(* Logix 5000 project; controller inz_PD_LK vendor 1 type 14 code 285 rev 34.11; software revision 34.01 *)

TASK MainTask (continuous, watchdog 500 ms) : Paleczka_silnik, Dzwonki_silnik, Paleczka_note_move, Dzwonki_belt_move, buttons, status, TIMER, Lights, oda, kolejnosc, dzwieki

MODULES
   Local : vendor 1 type 14 code 285 (5069 0, rev 34.11)
      serwowzmacniacz : vendor 1 type 45 code 1 (Ethernet 192.168.1.26, rev 5.2, AMotionDiagnostics RPI 1 ms)
      serwowzmacniacz2 : vendor 1 type 45 code 1 (Ethernet 192.168.1.27, rev 5.2, AMotionDiagnostics RPI 1 ms)
      Input : 5069-IB16 (5069 1, rev 2.1, StandardDataDriven RPI 5 ms)
      Output : 5069-OB16 (5069 2, rev 3.1, StandardDataDriven RPI 5 ms)
      Wyspa : 1734-AENTR (Ethernet 192.168.1.24, rev 5.12, Output RPI 20 ms)
         IB8 : 1734-IB8 (PointIO 3, rev 3.1)
         IB8_2 : 1734-IB8 (PointIO 4, rev 3.1)
         IE8C : vendor 1 type 115 code 210 (PointIO 6, rev 3.1, Input RPI 80 ms)
         OB8 : 1734-OB8 (PointIO 1, rev 3.1)
         OB8_2 : 1734-OB8 (PointIO 2, rev 3.1)
         OE4C : vendor 1 type 115 code 211 (PointIO 5, rev 3.1, Output RPI 80 ms)
END_MODULES

VAR_GLOBAL   (* controller tags *)
   all_rise : BOOL;
   auto_belt : BOOL;
   auto_mode : ALIAS FOR Local:1:I.Pt09.Data;
   auto_note : BOOL;
   belt_degree : DINT := 58;
   belt_finish : BOOL;
   D_JOG_Axis_OFF : BOOL := 1;
   D_JOG_Axis_ON : BOOL;
   D_motor_start : BOOL;
   D_motor_stop : BOOL := 1;
   degree : DINT := 20;
   dzwiek : DINT[50] := ([1] := 29, [2] := 29, [4] := -29, [5] := -29, [6] := -29, [7] := -29, [9] := 29, [10] := 29, [12] := -29, [14] := 29, [16] := 29, [17] := 29, [19] := -29, [20] := -29, [21] := -29, [22] := -29, [24] := 29, [25] := 29, [26] := -29, [27] := -29);
   Dzwonki : AXIS_CIP_DRIVE;
   Estop_button : ALIAS FOR Local:1:I.Pt00.Data;
   forced_OFF : BOOL;
   forced_ON : BOOL := 1;
   go_down : BOOL;
   go_left : ALIAS FOR Wyspa:3:I.5;
   go_right : ALIAS FOR Local:1:I.Pt02.Data;
   go_up : BOOL;
   green_lamp : ALIAS FOR Local:2:O.Pt13.Data;
   L_R_switch : ALIAS FOR Local:1:I.Pt10.Data;
   Motion : MOTION_GROUP;
   MotionControlMAFR_D : MOTION_INSTRUCTION := (FLAGS := 570425344, DN := 1, STATE := 1);
   MotionControlMAFR_P : MOTION_INSTRUCTION := (FLAGS := 570425344, DN := 1, STATE := 1);
   MotionControlMAH : MOTION_INSTRUCTION := (FLAGS := 33554432);
   MotionControlMAJ_P : MOTION_INSTRUCTION := (FLAGS := 301989888, ER := 1, ERR := 5);
   MotionControlMAM : MOTION_INSTRUCTION := (FLAGS := 570425344, DN := 1);
   MotionControlMAM2 : MOTION_INSTRUCTION := (FLAGS := 704643072, DN := 1, PC := 1);
   MotionControlMAM3 : MOTION_INSTRUCTION := (FLAGS := 704643072, DN := 1, PC := 1);
   MotionControlMAM4 : MOTION_INSTRUCTION := (FLAGS := 33554432);
   MotionControlMAM5 : MOTION_INSTRUCTION := (FLAGS := 704643072, DN := 1, PC := 1);
   MotionControlMAS_D : MOTION_INSTRUCTION := (FLAGS := -1442840576, EN := 1, DN := 1, PC := 1);
   MotionControlMAS_P : MOTION_INSTRUCTION := (FLAGS := -1442840576, EN := 1, DN := 1, PC := 1);
   MotionControlOFF_D : MOTION_INSTRUCTION := (FLAGS := -1577058304, EN := 1, DN := 1, STATUS := 2, STATE := 1);
   MotionControlOFF_P : MOTION_INSTRUCTION := (FLAGS := -1577058304, EN := 1, DN := 1, STATUS := 2, STATE := 1);
   MotionControlON_D : MOTION_INSTRUCTION := (FLAGS := 570425344, DN := 1, STATE := 1);
   MotionControlON_P : MOTION_INSTRUCTION := (FLAGS := 570425344, DN := 1, STATE := 1);
   move_belt : BOOL;
   neg_belt_degree : DINT := -58;
   neg_degree : INT := -20;
   OSR_auto_belt : BOOL;
   OSR_auto_note : BOOL;
   OSR_belt_ready : BOOL;
   OSR_D_motor_start : BOOL;
   OSR_D_motor_stop : BOOL;
   OSR_forced_OFF : BOOL;
   OSR_forced_ON : BOOL;
   OSR_moved : BOOL;
   OSR_P_motor_start : BOOL;
   OSR_P_motor_stop : BOOL;
   OSR_start_now : BOOL;
   OSR_starting_ON : BOOL;
   P_JOG_Axis_OFF : BOOL := 1;
   P_JOG_Axis_ON : BOOL;
   P_motor_start : BOOL;
   P_motor_stop : BOOL := 1;
   Paleczka : AXIS_CIP_DRIVE;
   play_note : BOOL;
   play_note_rise : BOOL;
   PULSE_1Hz : BOOL := 1;
   PULSE_2Hz : BOOL := 1;
   ready : BOOL;
   red_lamp : ALIAS FOR Local:2:O.Pt15.Data;
   reset : BOOL;
   reset_button : ALIAS FOR Local:1:I.Pt07.Data;
   stand_by : BOOL;
   start : BOOL; {access None}
   start_button : ALIAS FOR Local:1:I.Pt05.Data;
   start_degree : DINT := 20;
   start_now : BOOL;
   starting_ON : BOOL := 1;
   stop : BOOL := 1; {access None}
   switch_OFF : ALIAS FOR Local:1:I.Pt08.Data;
   switch_ON : ALIAS FOR Local:1:I.Pt09.Data;
   TIMER1N : TIMER := (PRE := 100);
   TIMER2N : TIMER := (PRE := 200);
   uderzenie : DINT[50] := ([0] := 20, [1] := 20, [2] := 20, [3] := 20, [4] := 20, [5] := 20);
   yellow_lamp : ALIAS FOR Local:2:O.Pt14.Data;
END_VAR

PROGRAM buttons   (* main routine buttons *)

ROUTINE buttons   (* ladder *)
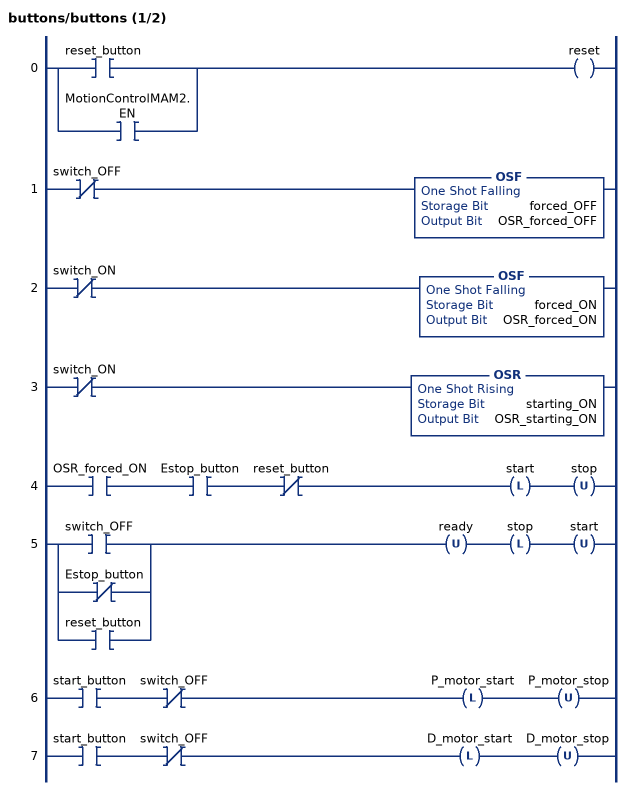
   0: [XIC(reset_button) ,XIC(MotionControlMAM2.EN) ]OTE(reset);
   1: XIO(switch_OFF)OSF(forced_OFF,OSR_forced_OFF);
   2: XIO(switch_ON)OSF(forced_ON,OSR_forced_ON);
   3: XIO(switch_ON)OSR(starting_ON,OSR_starting_ON);
   4: XIC(OSR_forced_ON)XIC(Estop_button)XIO(reset_button)OTL(start)OTU(stop);
   5: [XIC(switch_OFF) ,[XIO(Estop_button) ,XIC(reset_button) ] ]OTU(ready)OTL(stop)OTU(start);
   6: XIC(start_button)XIO(switch_OFF)OTL(P_motor_start)OTU(P_motor_stop);
   7: XIC(start_button)XIO(switch_OFF)OTL(D_motor_start)OTU(D_motor_stop);
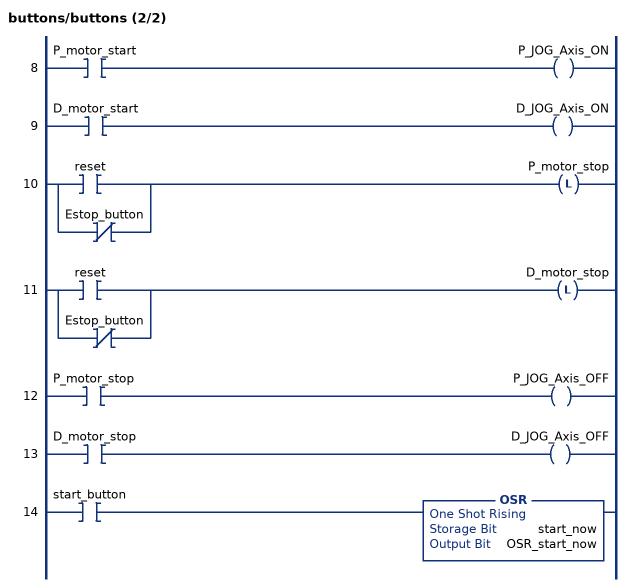
   8: XIC(P_motor_start)OTE(P_JOG_Axis_ON);
   9: XIC(D_motor_start)OTE(D_JOG_Axis_ON);
   10: [XIC(reset) ,XIO(Estop_button) ]OTL(P_motor_stop);
   11: [XIC(reset) ,XIO(Estop_button) ]OTL(D_motor_stop);
   12: XIC(P_motor_stop)OTE(P_JOG_Axis_OFF);
   13: XIC(D_motor_stop)OTE(D_JOG_Axis_OFF);
   14: XIC(start_button)OSR(start_now,OSR_start_now);
END_ROUTINE
END_PROGRAM

PROGRAM dzwieki   (* main routine dzwieki *)

ROUTINE dzwieki   (* structured text *)
   // "Oda do radości" zaczynając od E
   dzwiek[0] := 0;    //E <- druga nuta
   dzwiek[1] := 29;   //F
   dzwiek[2] := 29;   //G
   dzwiek[3] := 0;    //G
   dzwiek[4] := -29;  //F
   dzwiek[5] := -29;  //E
   dzwiek[6] := -29;  //D
   dzwiek[7] := -29;  //C
   dzwiek[8] := 0;    //C
   dzwiek[9] := 29;   //D
   dzwiek[10] := 29;  //E
   dzwiek[11] := 0;   //E
   dzwiek[12] := -29; //D
   dzwiek[13] := 0;   //D
   dzwiek[14] := 29;  //E
   dzwiek[15] := 0;   //E
   dzwiek[16] := 29;  //F
   dzwiek[17] := 29;  //G
   dzwiek[18] := 0;   //G
   dzwiek[19] := -29; //F
   dzwiek[20] := -29; //E
   dzwiek[21] := -29; //D
   dzwiek[22] := -29; //C
   dzwiek[23] := 0;   //C
   dzwiek[24] := 29;  //D
   dzwiek[25] := 29;  //E
   dzwiek[26] := -29; //D
   dzwiek[27] := -29; //C
   dzwiek[28] := 0;   //C
END_ROUTINE
END_PROGRAM

PROGRAM Dzwonki_belt_move   (* main routine belt_move *)
VAR
   acc : DINT := 2000;
   belt_moving : DINT := 30;
   belt_ready : BOOL;
   CTU1 : COUNTER := (ACC := 30, DN := 1);
   jerk : DINT := 14;
   odl : DINT := 58;
   speed : DINT := 10000;
END_VAR

ROUTINE belt_move   (* ladder *)
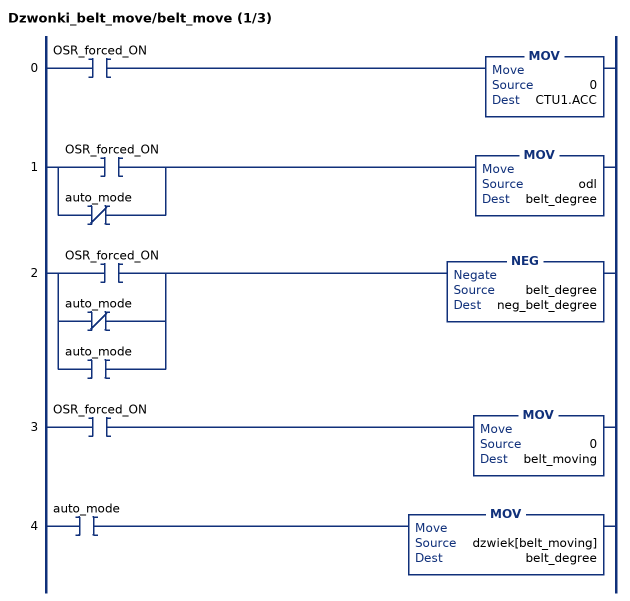
   0: XIC(OSR_forced_ON)MOV(0,CTU1.ACC);
   1: [XIC(OSR_forced_ON) ,XIO(auto_mode) ]MOV(odl,belt_degree);
   2: [XIC(OSR_forced_ON) ,[XIO(auto_mode) ,XIC(auto_mode) ] ]NEG(belt_degree,neg_belt_degree);
   3: XIC(OSR_forced_ON)MOV(0,belt_moving);
   4: XIC(auto_mode)MOV(dzwiek[belt_moving],belt_degree);
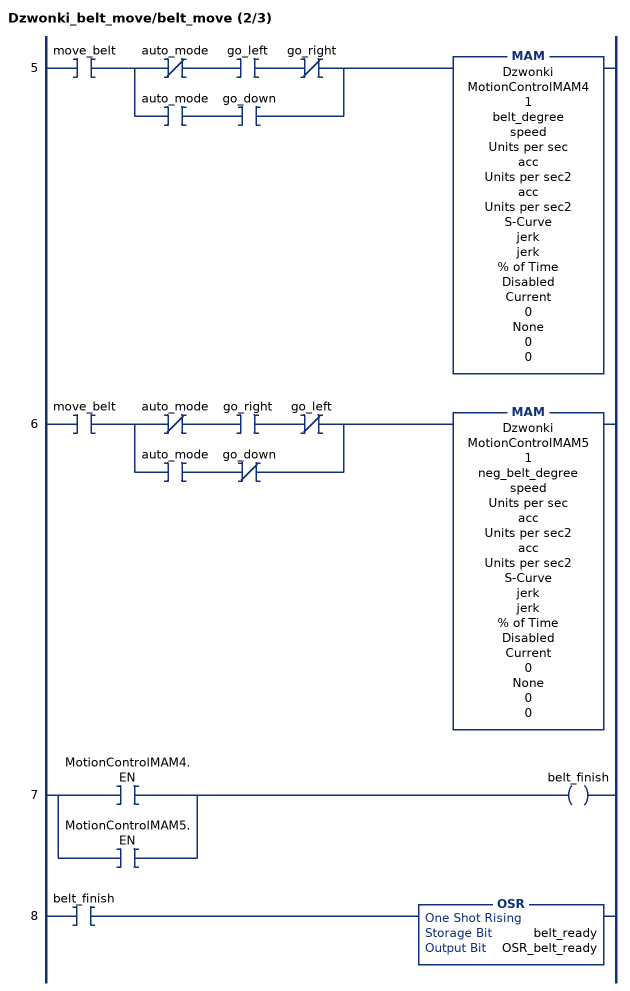
   5: XIC(move_belt)[XIO(auto_mode) XIC(go_left) XIO(go_right) ,XIC(auto_mode) XIC(go_down) ]MAM(Dzwonki,MotionControlMAM4,1,belt_degree,speed,Units per sec,acc,Units per sec2,acc,Units per sec2,S-Curve,jerk,jerk,% of Time,Disabled,Current,0,None,0,0);
   6: XIC(move_belt)[XIO(auto_mode) XIC(go_right) XIO(go_left) ,XIC(auto_mode) XIO(go_down) ]MAM(Dzwonki,MotionControlMAM5,1,neg_belt_degree,speed,Units per sec,acc,Units per sec2,acc,Units per sec2,S-Curve,jerk,jerk,% of Time,Disabled,Current,0,None,0,0);
   7: [XIC(MotionControlMAM4.EN) ,XIC(MotionControlMAM5.EN) ]OTE(belt_finish);
   8: XIC(belt_finish)OSR(belt_ready,OSR_belt_ready);
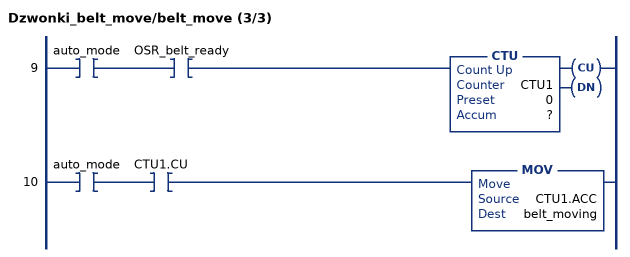
   9: XIC(auto_mode)XIC(OSR_belt_ready)CTU(CTU1,?,?);
   10: XIC(auto_mode)XIC(CTU1.CU)MOV(CTU1.ACC,belt_moving);
END_ROUTINE
END_PROGRAM

PROGRAM Dzwonki_silnik   (* main routine MainRoutine *)

ROUTINE MainRoutine   (* ladder *)
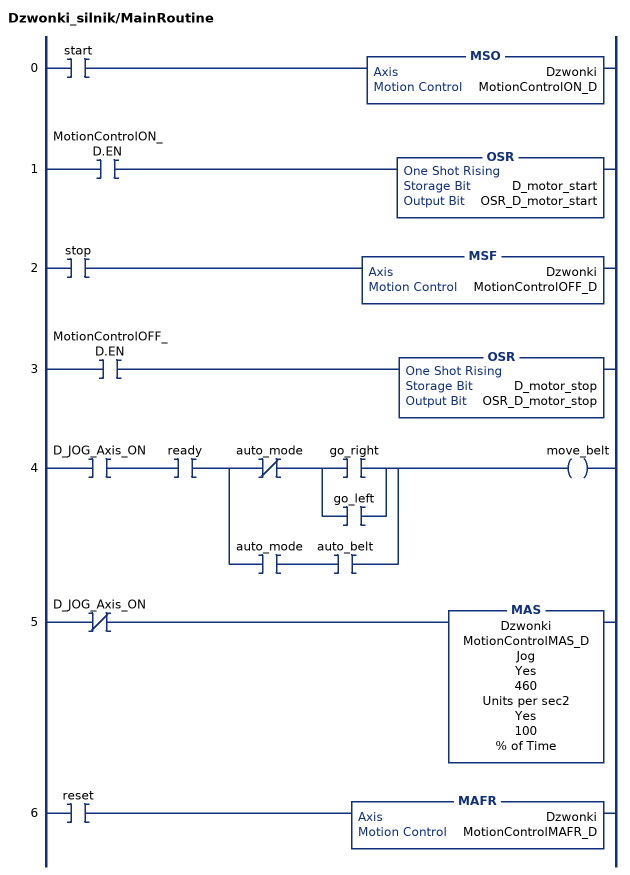
   0: XIC(start)MSO(Dzwonki,MotionControlON_D);
   1: XIC(MotionControlON_D.EN)OSR(D_motor_start,OSR_D_motor_start);
   2: XIC(stop)MSF(Dzwonki,MotionControlOFF_D);
   3: XIC(MotionControlOFF_D.EN)OSR(D_motor_stop,OSR_D_motor_stop);
   4: XIC(D_JOG_Axis_ON)XIC(ready)[XIO(auto_mode) [XIC(go_right) ,XIC(go_left) ] ,XIC(auto_mode) XIC(auto_belt) ]OTE(move_belt);
   5: XIO(D_JOG_Axis_ON)MAS(Dzwonki,MotionControlMAS_D,Jog,Yes,460,Units per sec2,Yes,100,% of Time);
   6: XIC(reset)MAFR(Dzwonki,MotionControlMAFR_D);
END_ROUTINE
END_PROGRAM

PROGRAM kolejnosc   (* main routine kolejnosc *)

ROUTINE kolejnosc   (* structured text *)
   uderzenie[0] := 20;
   uderzenie[1] := 20;
   uderzenie[2] := 20;
   uderzenie[3] := 20;
   uderzenie[4] := 20;
   uderzenie[5] := 20;
   
END_ROUTINE
END_PROGRAM

PROGRAM Lights   (* main routine Lights *)
VAR
   OSR_yellow_ON : BOOL;
   yellow_ON : BOOL;
END_VAR

ROUTINE Lights   (* ladder *)
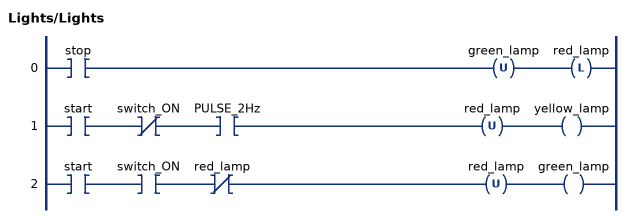
   0: XIC(stop)OTU(green_lamp)OTL(red_lamp);
   1: XIC(start)XIO(switch_ON)XIC(PULSE_2Hz)OTU(red_lamp)OTE(yellow_lamp);
   2: XIC(start)XIC(switch_ON)XIO(red_lamp)OTU(red_lamp)OTE(green_lamp);
END_ROUTINE
END_PROGRAM

PROGRAM oda   (* main routine oda *)
VAR
   CTU1 : COUNTER := (PRE := 1, ACC := 30, CD := 1, DN := 1);
   CTU1_CU : BOOL;
   CTU2 : COUNTER := (PRE := 5);
   even_odd : DINT;
   is_finished : BOOL;
   LCONS_INIT : INT;
   ONS_auto_belt : BOOL;
   ONS_auto_note : BOOL;
   ONS_is_finished : BOOL;
   OSR_CTU1_CU : BOOL;
   OSR_timer1_ready : BOOL;
   OSR_timer2_ready : BOOL;
   repeats : DINT;
   STEP : INT;
   timer1_ready : BOOL;
   TIMER1O : TIMER := (PRE := 100);
   timer2_ready : BOOL;
   TIMER2O : TIMER := (PRE := 100);
   TON1 : TIMER := (PRE := 50);
END_VAR

ROUTINE oda   (* ladder *)
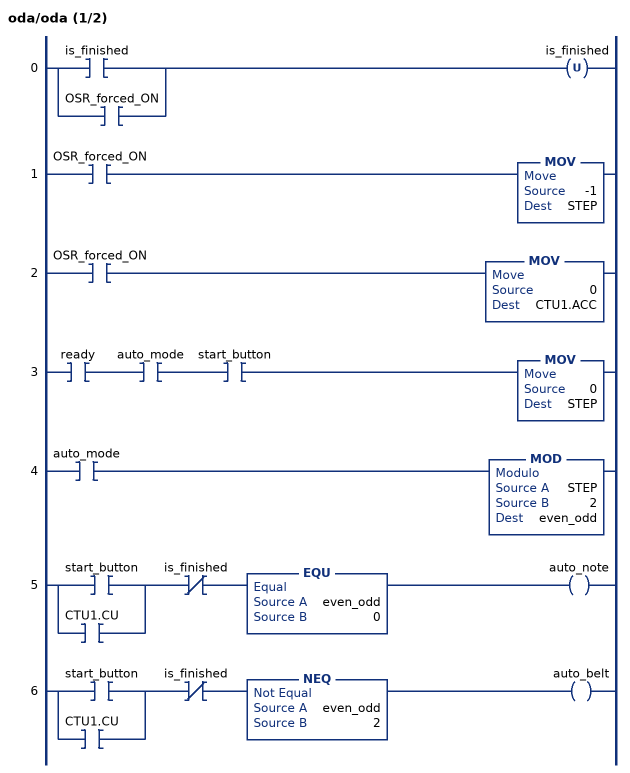
   0: [XIC(is_finished) ,XIC(OSR_forced_ON) ]OTU(is_finished);
   1: XIC(OSR_forced_ON)MOV(-1,STEP);
   2: XIC(OSR_forced_ON)MOV(0,CTU1.ACC);
   3: XIC(ready)XIC(auto_mode)XIC(start_button)MOV(0,STEP);
   4: XIC(auto_mode)MOD(STEP,2,even_odd);
   5: [XIC(start_button) ,XIC(CTU1.CU) ]XIO(is_finished)EQU(even_odd,0)OTE(auto_note);
   6: [XIC(start_button) ,XIC(CTU1.CU) ]XIO(is_finished)NEQ(even_odd,2)OTE(auto_belt);
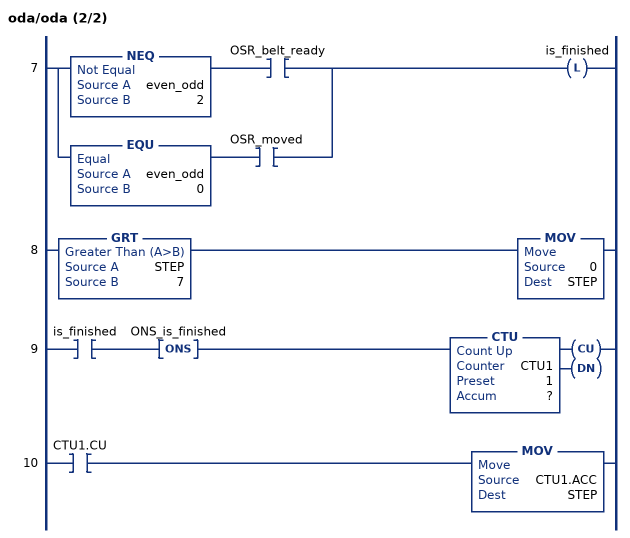
   7: [NEQ(even_odd,2) XIC(OSR_belt_ready) ,EQU(even_odd,0) XIC(OSR_moved) ]OTL(is_finished);
   8: GRT(STEP,7)MOV(0,STEP);
   9: XIC(is_finished)ONS(ONS_is_finished)CTU(CTU1,?,?);
   10: XIC(CTU1.CU)MOV(CTU1.ACC,STEP);
END_ROUTINE
END_PROGRAM

PROGRAM Paleczka_note_move   (* main routine note_move *)
VAR
   CTU1 : COUNTER := (DN := 1);
   moved : BOOL := 1;
   note_playing : DINT;
   ONS_note : BOOL;
   set_degree : DINT := -20;
   tone : DINT := -20;
END_VAR

ROUTINE note_move   (* ladder *)
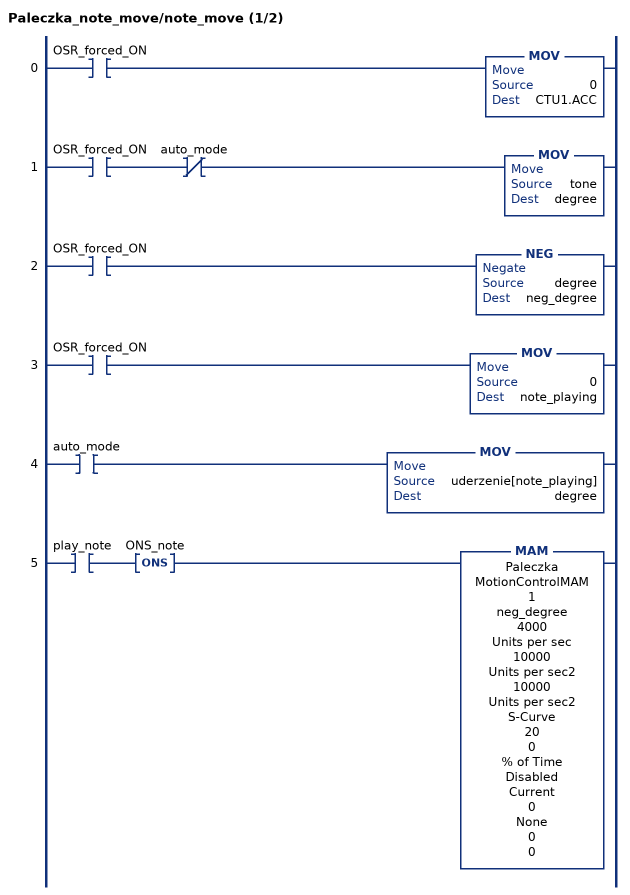
   0: XIC(OSR_forced_ON)MOV(0,CTU1.ACC);
   1: XIC(OSR_forced_ON)XIO(auto_mode)MOV(tone,degree);
   2: XIC(OSR_forced_ON)NEG(degree,neg_degree);
   3: XIC(OSR_forced_ON)MOV(0,note_playing);
   4: XIC(auto_mode)MOV(uderzenie[note_playing],degree);
   5: XIC(play_note)ONS(ONS_note)MAM(Paleczka,MotionControlMAM,1,neg_degree,4000,Units per sec,10000,Units per sec2,10000,Units per sec2,S-Curve,20,0,% of Time,Disabled,Current,0,None,0,0);
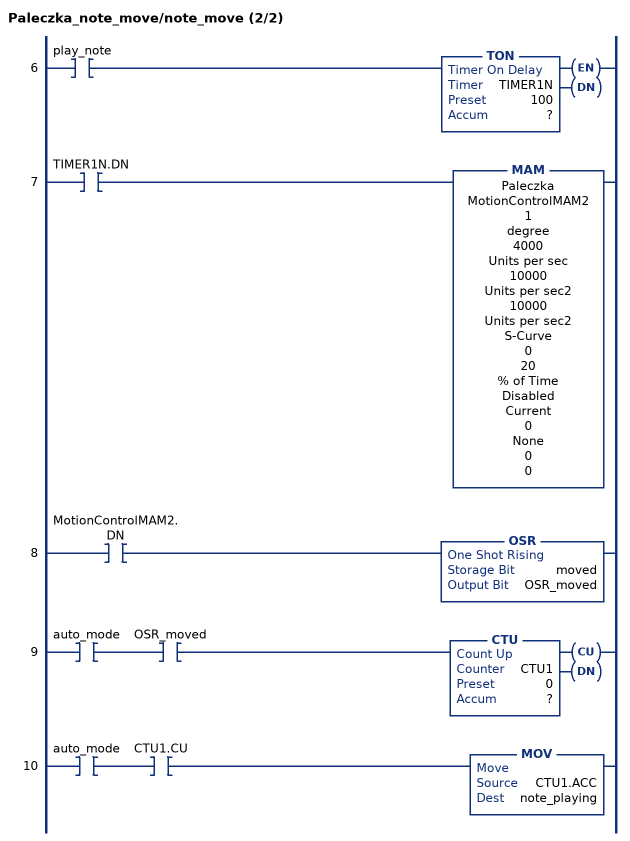
   6: XIC(play_note)TON(TIMER1N,?,?);
   7: XIC(TIMER1N.DN)MAM(Paleczka,MotionControlMAM2,1,degree,4000,Units per sec,10000,Units per sec2,10000,Units per sec2,S-Curve,0,20,% of Time,Disabled,Current,0,None,0,0);
   8: XIC(MotionControlMAM2.DN)OSR(moved,OSR_moved);
   9: XIC(auto_mode)XIC(OSR_moved)CTU(CTU1,?,?);
   10: XIC(auto_mode)XIC(CTU1.CU)MOV(CTU1.ACC,note_playing);
END_ROUTINE
END_PROGRAM

PROGRAM Paleczka_silnik   (* main routine MainRoutine *)

ROUTINE MainRoutine   (* ladder *)
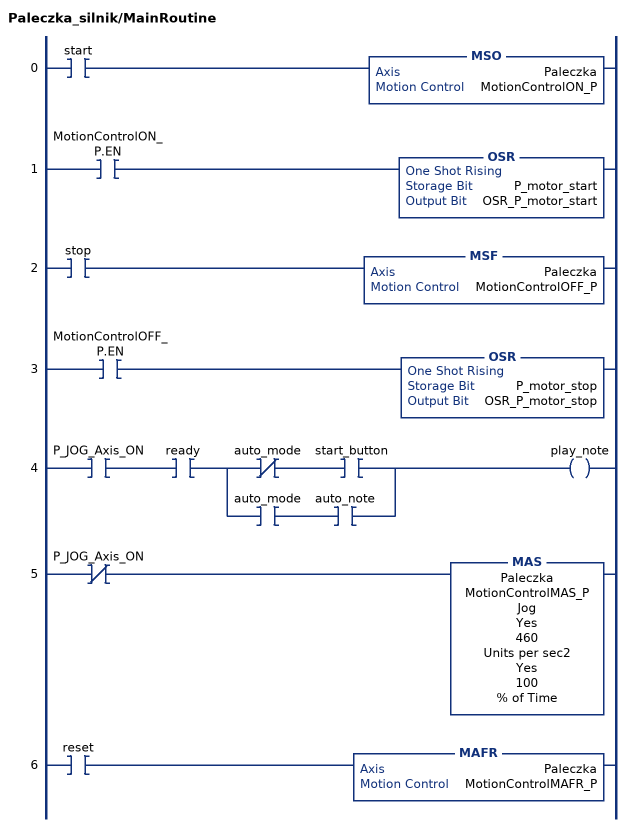
   0: XIC(start)MSO(Paleczka,MotionControlON_P);
   1: XIC(MotionControlON_P.EN)OSR(P_motor_start,OSR_P_motor_start);
   2: XIC(stop)MSF(Paleczka,MotionControlOFF_P);
   3: XIC(MotionControlOFF_P.EN)OSR(P_motor_stop,OSR_P_motor_stop);
   4: XIC(P_JOG_Axis_ON)XIC(ready)[XIO(auto_mode) XIC(start_button) ,XIC(auto_mode) XIC(auto_note) ]OTE(play_note);
   5: XIO(P_JOG_Axis_ON)MAS(Paleczka,MotionControlMAS_P,Jog,Yes,460,Units per sec2,Yes,100,% of Time);
   6: XIC(reset)MAFR(Paleczka,MotionControlMAFR_P);
END_ROUTINE
END_PROGRAM

PROGRAM status   (* main routine ready *)

ROUTINE ready   (* ladder *)
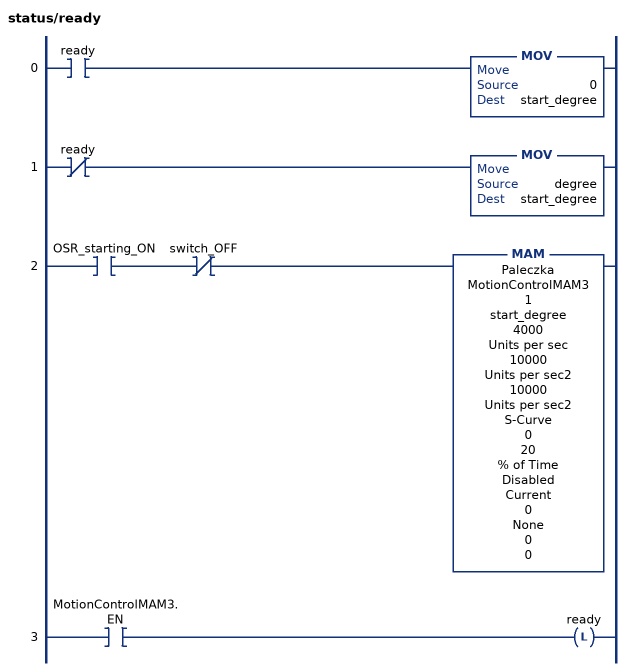
   0: XIC(ready)MOV(0,start_degree);
   1: XIO(ready)MOV(degree,start_degree);
   2: XIC(OSR_starting_ON)XIO(switch_OFF)MAM(Paleczka,MotionControlMAM3,1,start_degree,4000,Units per sec,10000,Units per sec2,10000,Units per sec2,S-Curve,0,20,% of Time,Disabled,Current,0,None,0,0);
   3: XIC(MotionControlMAM3.EN)OTL(ready);
END_ROUTINE
END_PROGRAM

PROGRAM TIMER   (* main routine pulse *)
VAR
   TIMER1 : TIMER := (PRE := 1000, ACC := 792, TT := 1, DN := 1);
   TIMER2 : TIMER := (PRE := 1000, ACC := 1000, EN := 1, DN := 1);
   TIMER3 : TIMER := (PRE := 500, ACC := 292, TT := 1, DN := 1);
   TIMER4 : TIMER := (PRE := 500, ACC := 500, EN := 1, DN := 1);
END_VAR

ROUTINE pulse   (* ladder *)
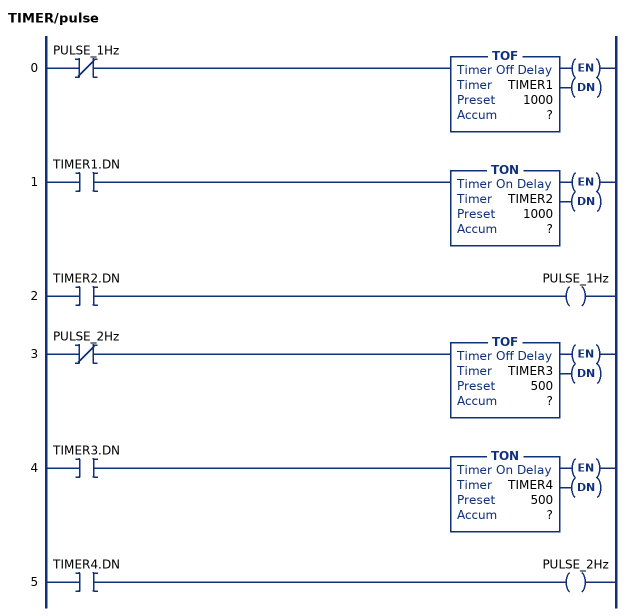
   0: XIO(PULSE_1Hz)TOF(TIMER1,?,?);
   1: XIC(TIMER1.DN)TON(TIMER2,?,?);
   2: XIC(TIMER2.DN)OTE(PULSE_1Hz);
   3: XIO(PULSE_2Hz)TOF(TIMER3,?,?);
   4: XIC(TIMER3.DN)TON(TIMER4,?,?);
   5: XIC(TIMER4.DN)OTE(PULSE_2Hz);
END_ROUTINE
END_PROGRAM
